KUKA KRL program: trigger2.src, trigger2.dat

--- trigger2.src ---
&ACCESS RVP
&REL 1
DEF  trigger2 ( )

  IF di004UseDryCycle==TRUE THEN

GOTO DRY
ELSE


IF  NUT_PRELOAD_STEP == 10 THEN
 ;HOME
;CL_QFPReturn / NUT FEED SLIDE RETURN
$OUT[503]=FALSE
$OUT[504]=TRUE
;dopw1_GUNHOME/VALVE2 OPEN
$OUT[472]=FALSE
$OUT[471]=TRUE
;CL_WeldPinRetract / UPPER PIN RETRACT
$OUT[498]=FALSE
$OUT[499]=TRUE
;CL_PartClampOpen
$OUT[501]=FALSE
$OUT[502]=TRUE
;CL_LowerPinExtend
$OUT[496]=FALSE
$OUT[495]=TRUE
$OUT[494]=TRUE
;QFP RETURNED
$OUT[503]=FALSE
$OUT[504]=TRUE
;CL_QFPAdvanced / QFP ADV
$OUT[504]=FALSE
$OUT[503]=TRUE
$OUT[476]=FALSE

IF ($IN[470]==TRUE) AND ($IN[482]==FALSE) THEN
   ;CL_QFPBlowOff / NUT FEED BLOW-OFF ACTIVATE
   $OUT[505]=TRUE
   ;CL_LowerPinRetreated
   $OUT[496]=FALSE
   $OUT[495]=TRUE
   NUT_PRELOAD_STEP = 20
   ELSE
ENDIF
ENDIF

ENDIF

   DRY:


END

--- trigger2.dat ---
&ACCESS RVP
&REL 1
DEFDAT  trigger2
;FOLD EXTERNAL DECLARATIONS;%{PE}%MKUKATPBASIS,%CEXT,%VCOMMON,%P
;FOLD BASISTECH EXT;%{PE}%MKUKATPBASIS,%CEXT,%VEXT,%P
EXT  BAS (BAS_COMMAND  :IN,REAL  :IN )
;ENDFOLD (BASISTECH EXT)
;FOLD USER EXT;%{E}%MKUKATPUSER,%CEXT,%VEXT,%P
;Make your modifications here

;ENDFOLD (USER EXT)
;ENDFOLD (EXTERNAL DECLARATIONS)
ENDDAT
